// TIA Portal project "Asansör Projesi" (V17)

(* hardware
DEVICE "S71500/ET200MP-Station_1"  S7-1500 station
   slot 0: "Profilschiene_0"  6ES7 590-1***0-0AA0
   slot 1: "PLC_1"  CPU 1511-1 PN  6ES7 511-1AK00-0AB0  V1.8
   slot 2: "AI 8xU/I/RTD/TC ST_1"  AI 8xU/I/RTD/TC ST  6ES7 531-7KF00-0AB0  V2.0
   slot 3: "AI 8xU/I/RTD/TC ST_2"  AI 8xU/I/RTD/TC ST  6ES7 531-7KF00-0AB0  V2.0
   slot 4: "AI 8xU/I/RTD/TC ST_3"  AI 8xU/I/RTD/TC ST  6ES7 531-7KF00-0AB0  V2.0
   slot 5: "AI 8xU/I/RTD/TC ST_4"  AI 8xU/I/RTD/TC ST  6ES7 531-7KF00-0AB0  V2.0
   slot 6: "DI 16x24VDC BA_1"  DI 16x24VDC BA  6ES7 521-1BH10-0AA0  V1.0
*)

// ===== PLC "PLC_1"  CPU 1511-1 PN =====

VAR_GLOBAL   // PLC tag table "Standard-Variablentabelle"
   "ŞALTER" AT %E0.0 : Bool;
   "ASANSÖR YUKARI" AT %A0.0 : Bool;
   "START" AT %E0.1 : Bool;
   "Tag_1" AT %M0.0 : Bool;
   "STOP" AT %I0.2 : Bool;
   "Tag_3" AT %I1.4 : Bool;
   "Tag_4" AT %M10.0 : Bool;
   "ASANSÖR AŞAĞI" AT %Q0.2 : Bool;
   "Tag_5" AT %I1.6 : Bool;
   "Tag_6" AT %I1.7 : Bool;
   "Tag_7" AT %M10.1 : Bool;
   "1.Konveyor" AT %Q0.5 : Bool;
   "SENSÖR 1" AT %I0.4 : Bool;
   "ASANSÖR YAVAŞLAMA" AT %Q0.1 : Bool;
   "Tag_8" AT %MD1 : DWord;
   "Tag_9" AT %MW10 : Int;
   "Tag_10" AT %ID38 : DWord;
   "DİF.SENSÖR 1" AT %I0.7 : Bool;
   "Tag_12" AT %M1.0 : Bool;
   "Tag_13" AT %M10.2 : Bool;
   "Tag_14" AT %M0.1 : Bool;
   "Tag_15" AT %I1.5 : Bool;
   "Tag_16" AT %M10.3 : Bool;
   "Tag_17" AT %M10.4 : Bool;
   "Tag_11" AT %M0.2 : Bool;
   "ASANSÖR GERİ" AT %Q0.4 : Bool;
   "Tag_19" AT %Q1.0 : Bool;
   "Tag_18" AT %Q0.3 : Bool;
   "Tag_20" AT %Q1.2 : Bool;
   "Tag_21" AT %Q0.6 : Bool;
   "Tag_22" AT %M0.3 : Bool;
   "Tag_23" AT %Q0.7 : Bool;
   "2.Konveyor" AT %Q1.1 : Bool;
   "Tag_25" AT %M10.5 : Bool;
   "Tag_26" AT %M10.6 : Bool;
   "Tag_27" AT %M10.7 : Bool;
   "Tag_2" AT %M0.4 : Bool;
   "Tag_28" AT %I1.2 : Bool;
   "Tag_29" AT %M11.0 : Bool;
   "Tag_30" AT %M11.1 : Bool;
   "Tag_31" AT %M11.2 : Bool;
   "Tag_32" AT %M11.3 : Bool;
   "DİF SENSÖR 2" AT %I1.0 : Bool;
   "SENSÖR 2" AT %I0.5 : Bool;
   "Tag_24" AT %M11.4 : Bool;
   "Tag_33" AT %M11.5 : Bool;
   "Tag_34" AT %M11.6 : Bool;
   "Tag_35" AT %M11.7 : Bool;
   "Tag_36" AT %M12.0 : Bool;
   "Tag_37" AT %M12.1 : Bool;
   "Tag_38" AT %M12.2 : Bool;
   "Tag_39" AT %I0.3 : Bool;
   "Tag_40" AT %M12.3 : Bool;
   "DIF SENSÖR 3" AT %I1.1 : Bool;
   "Tag_41" AT %M12.4 : Bool;
   "3.Konveyor" AT %Q1.3 : Bool;
   "SENSÖR 3" AT %I0.6 : Bool;
   "Tag_42" AT %M12.5 : Bool;
   "Tag_43" AT %M0.5 : Bool;
   "Asansör İleri" AT %Q1.4 : Bool;
   "Tag_44" AT %I1.3 : Bool;
   "Tag_45" AT %Q1.5 : Bool;
   "Tag_46" AT %I2.0 : Bool;
   "Tag_47" AT %M12.6 : Bool;
   "Tag_48" AT %M12.7 : Bool;
   "Tag_49" AT %M13.0 : Bool;
   "Tag_50" AT %M13.1 : Bool;
   "Tag_51" AT %M13.2 : Bool;
END_VAR

DATA_BLOCK "2.Kat_DB"   // DB4
{ S7_Optimized_Access := 'TRUE' }
VERSION : 0.1
// stored: InstanceOfName 2.Kat
"2.Kat"
BEGIN
END_DATA_BLOCK

DATA_BLOCK "1.Kat_DB"   // DB5
{ S7_Optimized_Access := 'TRUE' }
VERSION : 0.1
// stored: InstanceOfName 1.Kat
"1.Kat"
BEGIN
END_DATA_BLOCK

DATA_BLOCK "3.Kat_DB"   // DB10
{ S7_Optimized_Access := 'TRUE' }
VERSION : 0.1
// stored: InstanceOfName 3.Kat
"3.Kat"
BEGIN
END_DATA_BLOCK

// folder: System blocks/Program resources

DATA_BLOCK "IEC_Timer_0_DB"   // DB1
{ S7_Optimized_Access := 'TRUE' }
AUTHOR : Simatic
FAMILY : IEC
NAME : IEC_TMR
VERSION : 1.0
// stored: InstanceOfName IEC_TIMER
"IEC_TIMER"
BEGIN
END_DATA_BLOCK

DATA_BLOCK "IEC_Timer_0_DB_1"   // DB2
{ S7_Optimized_Access := 'TRUE' }
AUTHOR : Simatic
FAMILY : IEC
NAME : IEC_TMR
VERSION : 1.0
// stored: InstanceOfName IEC_TIMER
"IEC_TIMER"
BEGIN
END_DATA_BLOCK

DATA_BLOCK "IEC_Timer_0_DB_2"   // DB3
{ S7_Optimized_Access := 'TRUE' }
AUTHOR : Simatic
FAMILY : IEC
NAME : IEC_TMR
VERSION : 1.0
// stored: InstanceOfName IEC_TIMER
"IEC_TIMER"
BEGIN
END_DATA_BLOCK

DATA_BLOCK "IEC_Timer_0_DB_3"   // DB6
{ S7_Optimized_Access := 'TRUE' }
AUTHOR : Simatic
FAMILY : IEC
NAME : IEC_TMR
VERSION : 1.0
// stored: InstanceOfName IEC_TIMER
"IEC_TIMER"
BEGIN
END_DATA_BLOCK

DATA_BLOCK "IEC_Timer_0_DB_4"   // DB7
{ S7_Optimized_Access := 'TRUE' }
AUTHOR : Simatic
FAMILY : IEC
NAME : IEC_TMR
VERSION : 1.0
// stored: InstanceOfName IEC_TIMER
"IEC_TIMER"
BEGIN
END_DATA_BLOCK

DATA_BLOCK "IEC_Timer_0_DB_5"   // DB8
{ S7_Optimized_Access := 'TRUE' }
AUTHOR : Simatic
FAMILY : IEC
NAME : IEC_TMR
VERSION : 1.0
// stored: InstanceOfName IEC_TIMER
"IEC_TIMER"
BEGIN
END_DATA_BLOCK

DATA_BLOCK "IEC_Timer_0_DB_6"   // DB9
{ S7_Optimized_Access := 'TRUE' }
AUTHOR : Simatic
FAMILY : IEC
NAME : IEC_TMR
VERSION : 1.0
// stored: InstanceOfName IEC_TIMER
"IEC_TIMER"
BEGIN
END_DATA_BLOCK

// folder: (top level)

FUNCTION_BLOCK "1.Kat"   // FB1, LAD
{ S7_Optimized_Access := 'TRUE' }
VERSION : 0.1
   VAR_TEMP   // added for the SCL form of the ladder/FBD networks
      _w1 : Bool;
      _w2 : Bool;
      _w3 : Bool;
   END_VAR
BEGIN

REGION Network 1
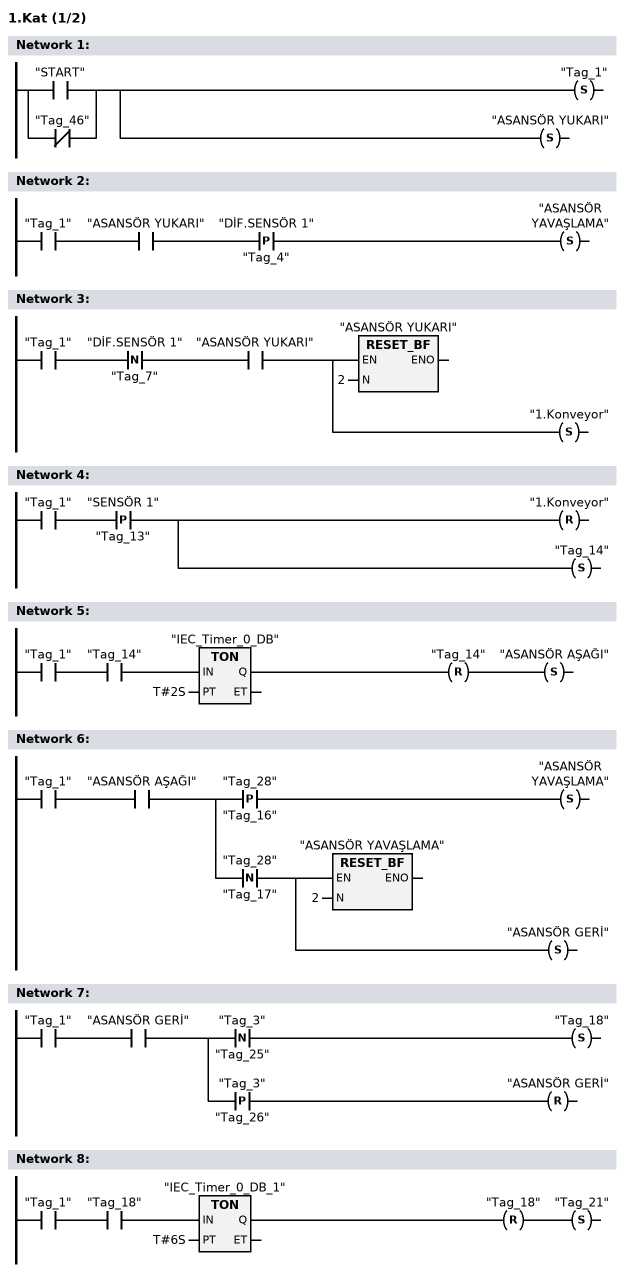
   RUNG wire#powerrail
      Contact( "START" )
      wire#w1
      S_Coil( "Tag_1" )
   END_RUNG
   RUNG wire#powerrail
      I_Contact( "Tag_46" )
   END_RUNG wire#w1
   RUNG wire#w1
      S_Coil( "ASANSÖR YUKARI" )
   END_RUNG
   // the same network as SCL:
   IF "START" OR NOT "Tag_46" THEN
       "Tag_1" := TRUE;
       "ASANSÖR YUKARI" := TRUE;
   END_IF;
END_REGION

REGION Network 2
   RUNG wire#powerrail
      Contact( "Tag_1" )
      Contact( "ASANSÖR YUKARI" )
      P_Contact(operand := "DİF.SENSÖR 1", bit := "Tag_4")
      S_Coil( "ASANSÖR YAVAŞLAMA" )
   END_RUNG
   // the same network as SCL:
   #_w1 := "Tag_1" AND "ASANSÖR YUKARI" AND "DİF.SENSÖR 1" AND NOT "Tag_4";   // rising edge of "DİF.SENSÖR 1"
   "Tag_4" := "DİF.SENSÖR 1";
   IF #_w1 THEN "ASANSÖR YAVAŞLAMA" := TRUE; END_IF;
END_REGION

REGION Network 3
   // no SCL statement known for RBitfield: written as a call
   #_w1 := "Tag_1" AND NOT "DİF.SENSÖR 1" AND "Tag_7";   // falling edge of "DİF.SENSÖR 1"
   "Tag_7" := "DİF.SENSÖR 1";
   #_w2 := #_w1 AND "ASANSÖR YUKARI";
   IF #_w2 THEN
       RESET_BF(operand := "ASANSÖR YUKARI", n := 2);
       "1.Konveyor" := TRUE;
   END_IF;
END_REGION

REGION Network 4
   RUNG wire#powerrail
      Contact( "Tag_1" )
      P_Contact(operand := "SENSÖR 1", bit := "Tag_13")
      wire#w1
      R_Coil( "1.Konveyor" )
   END_RUNG
   RUNG wire#w1
      S_Coil( "Tag_14" )
   END_RUNG
   // the same network as SCL:
   #_w1 := "Tag_1" AND "SENSÖR 1" AND NOT "Tag_13";   // rising edge of "SENSÖR 1"
   "Tag_13" := "SENSÖR 1";
   IF #_w1 THEN
       "1.Konveyor" := FALSE;
       "Tag_14" := TRUE;
   END_IF;
END_REGION

REGION Network 5
   "IEC_Timer_0_DB".TON(IN := "Tag_1" AND "Tag_14", PT := T#2S);
   IF "IEC_Timer_0_DB".Q THEN
       "Tag_14" := FALSE;
       "ASANSÖR AŞAĞI" := TRUE;
   END_IF;
END_REGION

REGION Network 6
   // no SCL statement known for RBitfield: written as a call
   #_w1 := "Tag_1" AND "ASANSÖR AŞAĞI";
   #_w2 := #_w1 AND "Tag_28" AND NOT "Tag_16";   // rising edge of "Tag_28"
   "Tag_16" := "Tag_28";
   IF #_w2 THEN "ASANSÖR YAVAŞLAMA" := TRUE; END_IF;
   #_w3 := #_w1 AND NOT "Tag_28" AND "Tag_17";   // falling edge of "Tag_28"
   "Tag_17" := "Tag_28";
   IF #_w3 THEN
       RESET_BF(operand := "ASANSÖR YAVAŞLAMA", n := 2);
       "ASANSÖR GERİ" := TRUE;
   END_IF;
END_REGION

REGION Network 7
   RUNG wire#powerrail
      Contact( "Tag_1" )
      Contact( "ASANSÖR GERİ" )
      wire#w1
      N_Contact(operand := "Tag_3", bit := "Tag_25")
      S_Coil( "Tag_18" )
   END_RUNG
   RUNG wire#w1
      P_Contact(operand := "Tag_3", bit := "Tag_26")
      R_Coil( "ASANSÖR GERİ" )
   END_RUNG
   // the same network as SCL:
   #_w1 := "Tag_1" AND "ASANSÖR GERİ";
   #_w2 := #_w1 AND NOT "Tag_3" AND "Tag_25";   // falling edge of "Tag_3"
   "Tag_25" := "Tag_3";
   IF #_w2 THEN "Tag_18" := TRUE; END_IF;
   #_w3 := #_w1 AND "Tag_3" AND NOT "Tag_26";   // rising edge of "Tag_3"
   "Tag_26" := "Tag_3";
   IF #_w3 THEN "ASANSÖR GERİ" := FALSE; END_IF;
END_REGION

REGION Network 8
   "IEC_Timer_0_DB_1".TON(IN := "Tag_1" AND "Tag_18", PT := T#6S);
   IF "IEC_Timer_0_DB_1".Q THEN
       "Tag_18" := FALSE;
       "Tag_21" := TRUE;
   END_IF;
END_REGION

REGION Network 9
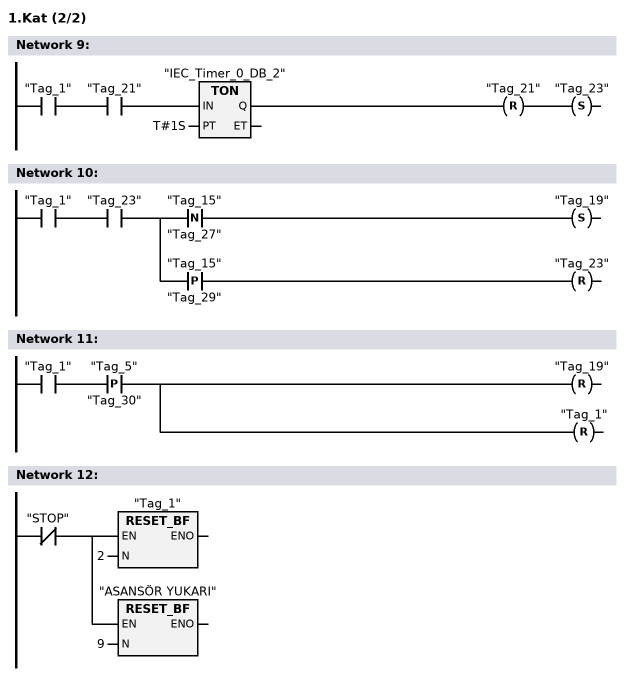
   "IEC_Timer_0_DB_2".TON(IN := "Tag_1" AND "Tag_21", PT := T#1S);
   IF "IEC_Timer_0_DB_2".Q THEN
       "Tag_21" := FALSE;
       "Tag_23" := TRUE;
   END_IF;
END_REGION

REGION Network 10
   RUNG wire#powerrail
      Contact( "Tag_1" )
      Contact( "Tag_23" )
      wire#w1
      N_Contact(operand := "Tag_15", bit := "Tag_27")
      S_Coil( "Tag_19" )
   END_RUNG
   RUNG wire#w1
      P_Contact(operand := "Tag_15", bit := "Tag_29")
      R_Coil( "Tag_23" )
   END_RUNG
   // the same network as SCL:
   #_w1 := "Tag_1" AND "Tag_23";
   #_w2 := #_w1 AND NOT "Tag_15" AND "Tag_27";   // falling edge of "Tag_15"
   "Tag_27" := "Tag_15";
   IF #_w2 THEN "Tag_19" := TRUE; END_IF;
   #_w3 := #_w1 AND "Tag_15" AND NOT "Tag_29";   // rising edge of "Tag_15"
   "Tag_29" := "Tag_15";
   IF #_w3 THEN "Tag_23" := FALSE; END_IF;
END_REGION

REGION Network 11
   RUNG wire#powerrail
      Contact( "Tag_1" )
      P_Contact(operand := "Tag_5", bit := "Tag_30")
      wire#w1
      R_Coil( "Tag_19" )
   END_RUNG
   RUNG wire#w1
      R_Coil( "Tag_1" )
   END_RUNG
   // the same network as SCL:
   #_w1 := "Tag_1" AND "Tag_5" AND NOT "Tag_30";   // rising edge of "Tag_5"
   "Tag_30" := "Tag_5";
   IF #_w1 THEN
       "Tag_19" := FALSE;
       "Tag_1" := FALSE;
   END_IF;
END_REGION

REGION Network 12
   // no SCL statement known for RBitfield: written as a call
   #_w1 := NOT "STOP";
   IF #_w1 THEN
       RESET_BF(operand := "Tag_1", n := 2);
       RESET_BF(operand := "ASANSÖR YUKARI", n := 9);
   END_IF;
END_REGION
END_FUNCTION_BLOCK

FUNCTION_BLOCK "2.Kat"   // FB2, LAD
{ S7_Optimized_Access := 'TRUE' }
VERSION : 0.1
   VAR_TEMP   // added for the SCL form of the ladder/FBD networks
      _w1 : Bool;
      _w2 : Bool;
      _w3 : Bool;
   END_VAR
BEGIN

REGION Network 1
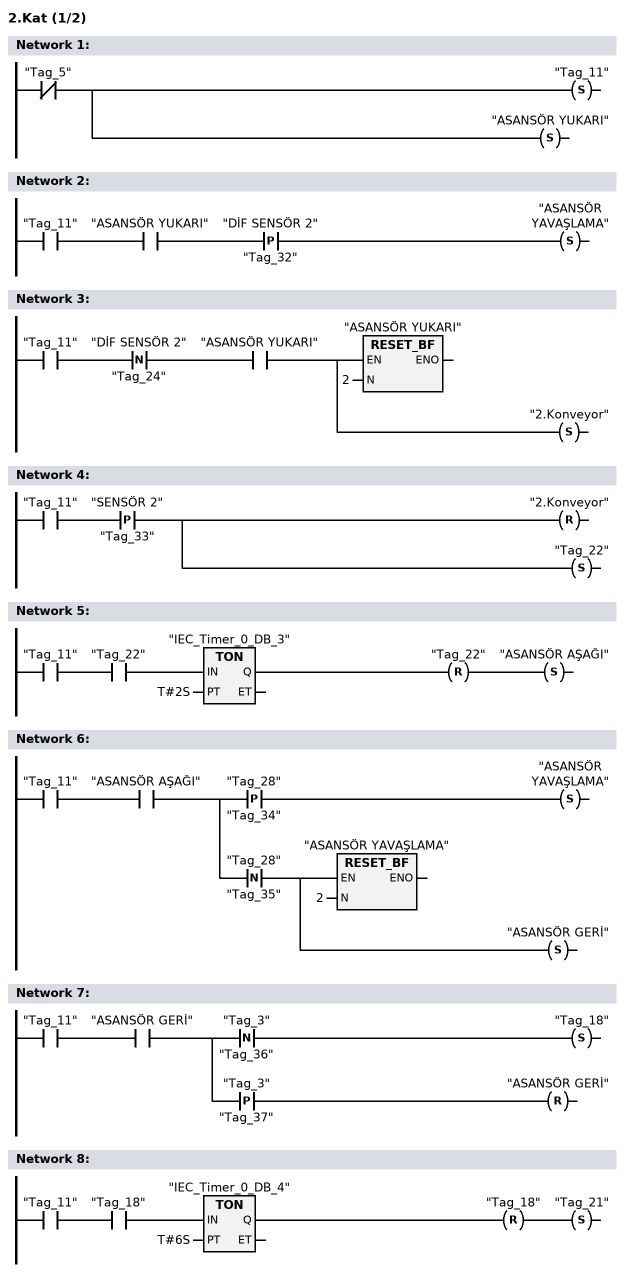
   RUNG wire#powerrail
      I_Contact( "Tag_5" )
      wire#w1
      S_Coil( "Tag_11" )
   END_RUNG
   RUNG wire#w1
      S_Coil( "ASANSÖR YUKARI" )
   END_RUNG
   // the same network as SCL:
   IF NOT "Tag_5" THEN
       "Tag_11" := TRUE;
       "ASANSÖR YUKARI" := TRUE;
   END_IF;
END_REGION

REGION Network 2
   RUNG wire#powerrail
      Contact( "Tag_11" )
      Contact( "ASANSÖR YUKARI" )
      P_Contact(operand := "DİF SENSÖR 2", bit := "Tag_32")
      S_Coil( "ASANSÖR YAVAŞLAMA" )
   END_RUNG
   // the same network as SCL:
   #_w1 := "Tag_11" AND "ASANSÖR YUKARI" AND "DİF SENSÖR 2" AND NOT "Tag_32";   // rising edge of "DİF SENSÖR 2"
   "Tag_32" := "DİF SENSÖR 2";
   IF #_w1 THEN "ASANSÖR YAVAŞLAMA" := TRUE; END_IF;
END_REGION

REGION Network 3
   // no SCL statement known for RBitfield: written as a call
   #_w1 := "Tag_11" AND NOT "DİF SENSÖR 2" AND "Tag_24";   // falling edge of "DİF SENSÖR 2"
   "Tag_24" := "DİF SENSÖR 2";
   #_w2 := #_w1 AND "ASANSÖR YUKARI";
   IF #_w2 THEN
       RESET_BF(operand := "ASANSÖR YUKARI", n := 2);
       "2.Konveyor" := TRUE;
   END_IF;
END_REGION

REGION Network 4
   RUNG wire#powerrail
      Contact( "Tag_11" )
      P_Contact(operand := "SENSÖR 2", bit := "Tag_33")
      wire#w1
      R_Coil( "2.Konveyor" )
   END_RUNG
   RUNG wire#w1
      S_Coil( "Tag_22" )
   END_RUNG
   // the same network as SCL:
   #_w1 := "Tag_11" AND "SENSÖR 2" AND NOT "Tag_33";   // rising edge of "SENSÖR 2"
   "Tag_33" := "SENSÖR 2";
   IF #_w1 THEN
       "2.Konveyor" := FALSE;
       "Tag_22" := TRUE;
   END_IF;
END_REGION

REGION Network 5
   "IEC_Timer_0_DB_3".TON(IN := "Tag_11" AND "Tag_22", PT := T#2S);
   IF "IEC_Timer_0_DB_3".Q THEN
       "Tag_22" := FALSE;
       "ASANSÖR AŞAĞI" := TRUE;
   END_IF;
END_REGION

REGION Network 6
   // no SCL statement known for RBitfield: written as a call
   #_w1 := "Tag_11" AND "ASANSÖR AŞAĞI";
   #_w2 := #_w1 AND "Tag_28" AND NOT "Tag_34";   // rising edge of "Tag_28"
   "Tag_34" := "Tag_28";
   IF #_w2 THEN "ASANSÖR YAVAŞLAMA" := TRUE; END_IF;
   #_w3 := #_w1 AND NOT "Tag_28" AND "Tag_35";   // falling edge of "Tag_28"
   "Tag_35" := "Tag_28";
   IF #_w3 THEN
       RESET_BF(operand := "ASANSÖR YAVAŞLAMA", n := 2);
       "ASANSÖR GERİ" := TRUE;
   END_IF;
END_REGION

REGION Network 7
   RUNG wire#powerrail
      Contact( "Tag_11" )
      Contact( "ASANSÖR GERİ" )
      wire#w1
      N_Contact(operand := "Tag_3", bit := "Tag_36")
      S_Coil( "Tag_18" )
   END_RUNG
   RUNG wire#w1
      P_Contact(operand := "Tag_3", bit := "Tag_37")
      R_Coil( "ASANSÖR GERİ" )
   END_RUNG
   // the same network as SCL:
   #_w1 := "Tag_11" AND "ASANSÖR GERİ";
   #_w2 := #_w1 AND NOT "Tag_3" AND "Tag_36";   // falling edge of "Tag_3"
   "Tag_36" := "Tag_3";
   IF #_w2 THEN "Tag_18" := TRUE; END_IF;
   #_w3 := #_w1 AND "Tag_3" AND NOT "Tag_37";   // rising edge of "Tag_3"
   "Tag_37" := "Tag_3";
   IF #_w3 THEN "ASANSÖR GERİ" := FALSE; END_IF;
END_REGION

REGION Network 8
   "IEC_Timer_0_DB_4".TON(IN := "Tag_11" AND "Tag_18", PT := T#6S);
   IF "IEC_Timer_0_DB_4".Q THEN
       "Tag_18" := FALSE;
       "Tag_21" := TRUE;
   END_IF;
END_REGION

REGION Network 9
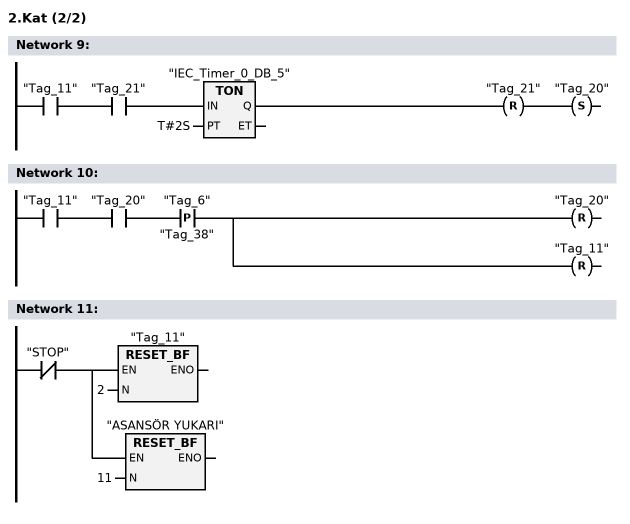
   "IEC_Timer_0_DB_5".TON(IN := "Tag_11" AND "Tag_21", PT := T#2S);
   IF "IEC_Timer_0_DB_5".Q THEN
       "Tag_21" := FALSE;
       "Tag_20" := TRUE;
   END_IF;
END_REGION

REGION Network 10
   RUNG wire#powerrail
      Contact( "Tag_11" )
      Contact( "Tag_20" )
      P_Contact(operand := "Tag_6", bit := "Tag_38")
      wire#w1
      R_Coil( "Tag_20" )
   END_RUNG
   RUNG wire#w1
      R_Coil( "Tag_11" )
   END_RUNG
   // the same network as SCL:
   #_w1 := "Tag_11" AND "Tag_20" AND "Tag_6" AND NOT "Tag_38";   // rising edge of "Tag_6"
   "Tag_38" := "Tag_6";
   IF #_w1 THEN
       "Tag_20" := FALSE;
       "Tag_11" := FALSE;
   END_IF;
END_REGION

REGION Network 11
   // no SCL statement known for RBitfield: written as a call
   #_w1 := NOT "STOP";
   IF #_w1 THEN
       RESET_BF(operand := "Tag_11", n := 2);
       RESET_BF(operand := "ASANSÖR YUKARI", n := 11);
   END_IF;
END_REGION
END_FUNCTION_BLOCK

FUNCTION_BLOCK "3.Kat"   // FB3, LAD
{ S7_Optimized_Access := 'TRUE' }
VERSION : 0.1
   VAR_TEMP   // added for the SCL form of the ladder/FBD networks
      _w1 : Bool;
      _w2 : Bool;
      _w3 : Bool;
   END_VAR
BEGIN

REGION Network 1
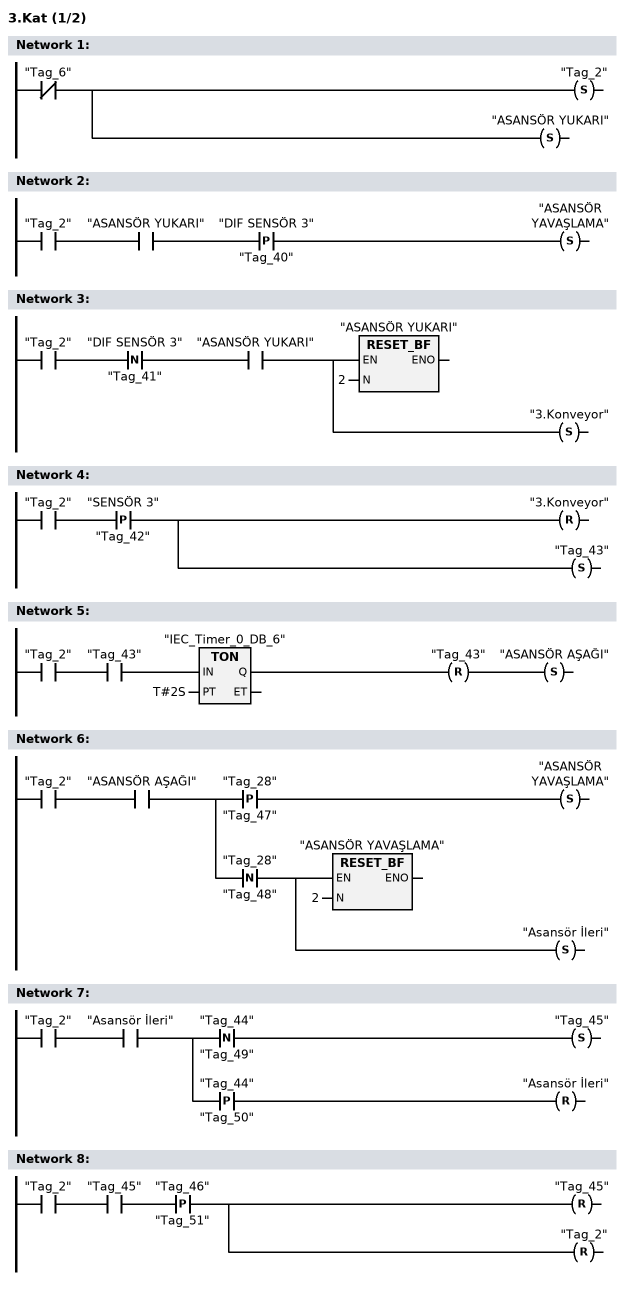
   RUNG wire#powerrail
      I_Contact( "Tag_6" )
      wire#w1
      S_Coil( "Tag_2" )
   END_RUNG
   RUNG wire#w1
      S_Coil( "ASANSÖR YUKARI" )
   END_RUNG
   // the same network as SCL:
   IF NOT "Tag_6" THEN
       "Tag_2" := TRUE;
       "ASANSÖR YUKARI" := TRUE;
   END_IF;
END_REGION

REGION Network 2
   RUNG wire#powerrail
      Contact( "Tag_2" )
      Contact( "ASANSÖR YUKARI" )
      P_Contact(operand := "DIF SENSÖR 3", bit := "Tag_40")
      S_Coil( "ASANSÖR YAVAŞLAMA" )
   END_RUNG
   // the same network as SCL:
   #_w1 := "Tag_2" AND "ASANSÖR YUKARI" AND "DIF SENSÖR 3" AND NOT "Tag_40";   // rising edge of "DIF SENSÖR 3"
   "Tag_40" := "DIF SENSÖR 3";
   IF #_w1 THEN "ASANSÖR YAVAŞLAMA" := TRUE; END_IF;
END_REGION

REGION Network 3
   // no SCL statement known for RBitfield: written as a call
   #_w1 := "Tag_2" AND NOT "DIF SENSÖR 3" AND "Tag_41";   // falling edge of "DIF SENSÖR 3"
   "Tag_41" := "DIF SENSÖR 3";
   #_w2 := #_w1 AND "ASANSÖR YUKARI";
   IF #_w2 THEN
       RESET_BF(operand := "ASANSÖR YUKARI", n := 2);
       "3.Konveyor" := TRUE;
   END_IF;
END_REGION

REGION Network 4
   RUNG wire#powerrail
      Contact( "Tag_2" )
      P_Contact(operand := "SENSÖR 3", bit := "Tag_42")
      wire#w1
      R_Coil( "3.Konveyor" )
   END_RUNG
   RUNG wire#w1
      S_Coil( "Tag_43" )
   END_RUNG
   // the same network as SCL:
   #_w1 := "Tag_2" AND "SENSÖR 3" AND NOT "Tag_42";   // rising edge of "SENSÖR 3"
   "Tag_42" := "SENSÖR 3";
   IF #_w1 THEN
       "3.Konveyor" := FALSE;
       "Tag_43" := TRUE;
   END_IF;
END_REGION

REGION Network 5
   "IEC_Timer_0_DB_6".TON(IN := "Tag_2" AND "Tag_43", PT := T#2S);
   IF "IEC_Timer_0_DB_6".Q THEN
       "Tag_43" := FALSE;
       "ASANSÖR AŞAĞI" := TRUE;
   END_IF;
END_REGION

REGION Network 6
   // no SCL statement known for RBitfield: written as a call
   #_w1 := "Tag_2" AND "ASANSÖR AŞAĞI";
   #_w2 := #_w1 AND "Tag_28" AND NOT "Tag_47";   // rising edge of "Tag_28"
   "Tag_47" := "Tag_28";
   IF #_w2 THEN "ASANSÖR YAVAŞLAMA" := TRUE; END_IF;
   #_w3 := #_w1 AND NOT "Tag_28" AND "Tag_48";   // falling edge of "Tag_28"
   "Tag_48" := "Tag_28";
   IF #_w3 THEN
       RESET_BF(operand := "ASANSÖR YAVAŞLAMA", n := 2);
       "Asansör İleri" := TRUE;
   END_IF;
END_REGION

REGION Network 7
   RUNG wire#powerrail
      Contact( "Tag_2" )
      Contact( "Asansör İleri" )
      wire#w1
      N_Contact(operand := "Tag_44", bit := "Tag_49")
      S_Coil( "Tag_45" )
   END_RUNG
   RUNG wire#w1
      P_Contact(operand := "Tag_44", bit := "Tag_50")
      R_Coil( "Asansör İleri" )
   END_RUNG
   // the same network as SCL:
   #_w1 := "Tag_2" AND "Asansör İleri";
   #_w2 := #_w1 AND NOT "Tag_44" AND "Tag_49";   // falling edge of "Tag_44"
   "Tag_49" := "Tag_44";
   IF #_w2 THEN "Tag_45" := TRUE; END_IF;
   #_w3 := #_w1 AND "Tag_44" AND NOT "Tag_50";   // rising edge of "Tag_44"
   "Tag_50" := "Tag_44";
   IF #_w3 THEN "Asansör İleri" := FALSE; END_IF;
END_REGION

REGION Network 8
   RUNG wire#powerrail
      Contact( "Tag_2" )
      Contact( "Tag_45" )
      P_Contact(operand := "Tag_46", bit := "Tag_51")
      wire#w1
      R_Coil( "Tag_45" )
   END_RUNG
   RUNG wire#w1
      R_Coil( "Tag_2" )
   END_RUNG
   // the same network as SCL:
   #_w1 := "Tag_2" AND "Tag_45" AND "Tag_46" AND NOT "Tag_51";   // rising edge of "Tag_46"
   "Tag_51" := "Tag_46";
   IF #_w1 THEN
       "Tag_45" := FALSE;
       "Tag_2" := FALSE;
   END_IF;
END_REGION

REGION Network 9
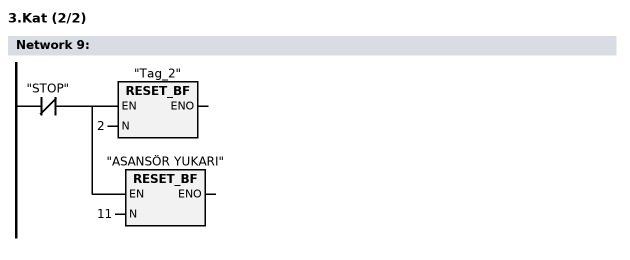
   // no SCL statement known for RBitfield: written as a call
   #_w1 := NOT "STOP";
   IF #_w1 THEN
       RESET_BF(operand := "Tag_2", n := 2);
       RESET_BF(operand := "ASANSÖR YUKARI", n := 11);
   END_IF;
END_REGION
END_FUNCTION_BLOCK

FUNCTION "MHJ-PLC-Lab-Function-S71500" : Void   // FC9000, SCL
{ S7_Optimized_Access := 'TRUE' }
VERSION : 0.1
   VAR_TEMP
      Value : Byte;
      ForCounter : Int;
   END_VAR
   VAR CONSTANT
      Value_01_DW : DWord := 16#1223_5486;
      Value_02_DW : DWord := 16#A6C9_D1F5;
   END_VAR
BEGIN

   #Value:=PEEK(area := 16#82,
        dbNumber := 0,
        byteOffset := 511);
   #Value := #Value + 1;

   POKE(area := 16#82,
        dbNumber := 0,
        byteOffset := 511,
        value := #Value);

   POKE(area := 16#82,
        dbNumber := 0,
        byteOffset := 1016,
        value := #Value_01_DW);
   POKE(area := 16#82,
        dbNumber := 0,
        byteOffset := 1020,
        value := #Value_02_DW);

   FOR #ForCounter := 0 TO 63 DO
       #Value:=PEEK(area := 16#1,
            dbNumber := 0,
            byteOffset := #ForCounter);
       POKE(area := 16#81,
            dbNumber := 0,
            byteOffset := #ForCounter,
            value := #Value);
   END_FOR;
   #Value := PEEK(area := 16#1,
                  dbNumber := 0,
                  byteOffset := 512);
   POKE(area := 16#82,
        dbNumber := 0,
        byteOffset := 512,
        value := #Value);
END_FUNCTION

ORGANIZATION_BLOCK "Main"   // OB1, LAD, ProgramCycle
TITLE = "Main Program Sweep (Cycle)"
{ S7_Optimized_Access := 'TRUE' }
VERSION : 0.1
   VAR_INPUT
      Initial_Call : Bool;   // Initial call of this OB
      Remanence : Bool;   // =True, if remanent data are available
   END_VAR
   VAR_TEMP   // added for the SCL form of the ladder/FBD networks
      _w1 : Bool;
      _w2 : Bool;
   END_VAR
BEGIN

REGION Network 1
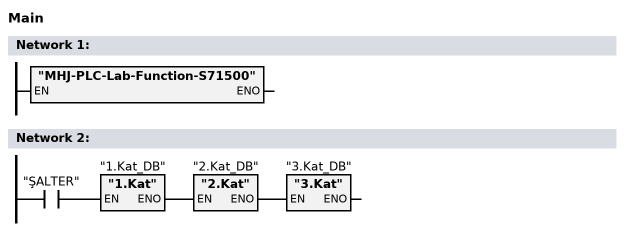
   RUNG wire#powerrail
      "MHJ-PLC-Lab-Function-S71500"()
   END_RUNG
   // the same network as SCL:
   "MHJ-PLC-Lab-Function-S71500"();
END_REGION

REGION Network 2
   RUNG wire#powerrail
      Contact( "ŞALTER" )
      "1.Kat_DB"()
      "2.Kat_DB"()
      "3.Kat_DB"()
   END_RUNG
   // the same network as SCL:
   "1.Kat_DB"(EN := "ŞALTER", ENO => #_w1);   // "1.Kat"
   "2.Kat_DB"(EN := #_w1, ENO => #_w2);   // "2.Kat"
   IF #_w2 THEN
       "3.Kat_DB"();   // "3.Kat"
   END_IF;
END_REGION
END_ORGANIZATION_BLOCK